// TIA Portal project "Project_Timers" (V16)

(* hardware
DEVICE "S7-1200 station_1"  S7-1200 Station
   slot 0: "Rack_0"  S7-1200 Rack  Rack  V1.0
   slot 1: "PLC_1"  CPU 1212C DC/DC/Rly  6ES7 212-1HE40-0XB0  V4.4
*)

// ===== PLC "PLC_1"  CPU 1212C DC/DC/Rly =====

VAR_GLOBAL   // PLC tag table "Default tag table"
   "START BUT" AT %I0.0 : Bool;
   "STOP BUT" AT %I0.1 : Bool;
   "MOTOR 1 KONT" AT %Q0.0 : Bool;
   "MOTOR 2 KONT" AT %Q0.1 : Bool;
   "MOTOR 3 KONT" AT %Q0.2 : Bool;
   "START MEM" AT %M30.0 : Bool;
END_VAR

// folder: System blocks/Program resources

DATA_BLOCK "TIMER 1"   // DB1
{ S7_Optimized_Access := 'TRUE' }
AUTHOR : Simatic
FAMILY : IEC
NAME : IEC_TMR
VERSION : 1.0
// stored: InstanceOfName IEC_TIMER
"IEC_TIMER"
BEGIN
END_DATA_BLOCK

// folder: (top level)

ORGANIZATION_BLOCK "Main"   // OB1, LAD, ProgramCycle
TITLE = "Main Program Sweep (Cycle)"
{ S7_Optimized_Access := 'TRUE' }
VERSION : 0.1
   VAR_INPUT
      Initial_Call : Bool;   // Initial call of this OB
      Remanence : Bool;   // =True, if remanent data are available
   END_VAR
BEGIN

REGION Network 1
   // Start butonuna basınca 1. ve 2. motor aynı anda calısacak, stop butonuna basınca tüm motorlar duracak.
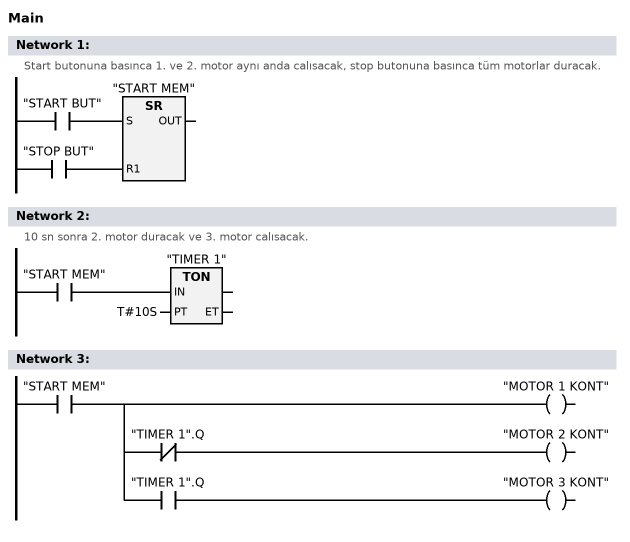
   RUNG wire#powerrail
      Contact( "START BUT" )
      S_SR(operand := "START MEM", r1 := wire#w1)
   END_RUNG
   RUNG wire#powerrail
      Contact( "STOP BUT" )
   END_RUNG wire#w1
   // the same network as SCL:
   IF "START BUT" THEN
       "START MEM" := TRUE;   // SR flip-flop
   END_IF;
   IF "STOP BUT" THEN "START MEM" := FALSE; END_IF;
END_REGION

REGION Network 2
   // 10 sn sonra 2. motor duracak ve 3. motor calısacak.
   "TIMER 1".TON(IN := "START MEM", PT := T#10S);
END_REGION

REGION Network 3
   RUNG wire#powerrail
      Contact( "START MEM" )
      wire#w1
      Coil( "MOTOR 1 KONT" )
   END_RUNG
   RUNG wire#w1
      I_Contact( "TIMER 1".Q )
      Coil( "MOTOR 2 KONT" )
   END_RUNG
   RUNG wire#w1
      Contact( "TIMER 1".Q )
      Coil( "MOTOR 3 KONT" )
   END_RUNG
   // the same network as SCL:
   "MOTOR 1 KONT" := "START MEM";
   "MOTOR 2 KONT" := "START MEM" AND NOT "TIMER 1".Q;
   "MOTOR 3 KONT" := "START MEM" AND "TIMER 1".Q;
END_REGION
END_ORGANIZATION_BLOCK